PROGRAM MAIN_simu
VAR
    simIO : MNG_Simulation;
END_VAR

// Update IOs with simulation
simIO(bEnable := TRUE);

// Application code follows here:

END_PROGRAM

(* stored: Version 1.1.0.1, ProductVersion 3.1.0.25
   POU MAIN_simu: Id {6437416a-b1ab-491b-b227-e4a8ab9af743} *)
